(*
Specifies the behaviour of :itf:`FB_Deadband` when the input is within the band.
*)
{attribute 'qualified_only'}
{attribute 'strict'}
{attribute 'to_string'}
TYPE E_DeadbandMode :
(
	Hold := 0, // Output holds its last value while the input is within the band.
	Zero := 1  // Output is set to zero while the input is within the band.
)BYTE;
END_TYPE

(* stored: Version 1.1.0.1, ProductVersion 3.1.4024.15
   EnumerationTextList E_DeadbandMode: Id {ff38a950-19ce-45a1-840d-1906b15948ac} *)
